PROGRAM Stn055_31_Stn411MainMergePrestop
VAR
	
	{attribute 'TcLinkToOSO' := '.iPuckPresent   :=  <0,1,2>TIIB[N67S00 (AL1332)]^N67S03 (AL2341)^TxPDO^input byte 0;
		.iBufferFull  :=  <0,1,2>TIIB[N67S00 (AL1332)]^N67S03 (AL2341)^TxPDO^input byte 2;
		.oStopLower :=  <0,1,1>TIIB[N67S00 (AL1332)]^N67S02 (EX260)^RxPDO^output byte 1'}
	fbConvStop: FB_ConvStop;
END_VAR

//  This code instantiates a component that is implimented as a common function block
//    Note that I/O is linked directly to I/O variables inside the named instance

gStn055_31_Stn411MainMergePrestop.ConvRunning := gConsumed_SafetyInterfaceConv.MtrRunning.Enc061Mtr04;

fbConvStop(
	pStn := ADR(gStn055),
	pCmp := ADR(gStn055_31_Stn411MainMergePrestop),
	pUpstreamStop := 0,
	pStateTraceBuffer := ADR(gStn055_StateTraceBuffer),
	pStateTraceFifo := ADR(gStn055_StateTraceFifo),
	pStats := ADR(gStn055_02_Stats));

END_PROGRAM

(* stored: Version 1.1.0.1, ProductVersion 3.1.4024.6
   POU Stn055_31_Stn411MainMergePrestop: Id {cc3ea658-7568-42d5-8205-3a4acd9ae1d6}, SpecialFunc None *)
